FUNCTION_BLOCK Fb_SafetyCheck
VAR_INPUT
END_VAR
VAR_OUTPUT
END_VAR
VAR
	i, j:INT;
	m_checkDelay :ARRAY[1..g_maxNum] OF checkDelay;
	m_checkDelayTime :checkDelayTime;
	m_checkPermit:ARRAY[1..g_maxNum] OF  checkPermit;
	
	m_jntErrFlag:ARRAY[1..g_maxNum,0..g_maxArmJoint,1..3] OF BOOL;
	m_armErrFlag:ARRAY [1..g_maxNum,1..3] OF BOOL;
	m_errCode:UDINT;
	
	
	m_errNumType: ARRAY [1..3] OF INT;
	m_ArrayErrCodeType:ARRAY [1..3] OF ARRAY [0..100] OF UDINT;
	
	//The fault is sent to the UI at the frequency of 0.1S
	m_errCodeUpdateFlag: ARRAY [1..3] OF BOOL;
	m_errCodeUpdateTon: ARRAY [1..3] OF TON;
	
	m_curJntTorqueIOlast :ARRAY [1..g_maxArmNum] OF vec7di;  
	m_cmdJntPosLast : ARRAY [1..g_maxArmNum] OF vec7d;  
	m_cartCurJntTorqueIOlast :ARRAY [1..4] OF LREAL;  
	m_cartCmdJntPosLast : ARRAY [1..4] OF LREAL; 
	o_ErrCode:ARRAY [1..3] OF UDINT;
		
	m_PromptMassBusy:BOOL;
	m_PromptFlag:ARRAY[1..g_maxNum,1..20] OF UINT;
	m_deleteCode:UDINT;
	
END_VAR


VAR CONSTANT
	m_codeUpdateDelay:TIME:=T#0.1S;
	
	//Fault level: 1 indicates  prompt message, 2 indicates a recoverable fault and 3 indicates an unrecoverable fault
	m_promptMessageLevel : UINT :=1;
	m_rcvLevel : UINT :=2;
	m_unrcvLevel : UINT :=3;
END_VAR

METHOD armSafetyCheck : BOOL
VAR_INPUT
	i_armId:UDINT;
	i_safetyCheckVar :ARRAY[1..g_maxNum] OF checkInputVariable;
	i_masterJointData : ST_MasterJointData;
END_VAR

VAR
	k:INT;
END_VAR

//驱动器状态监测、驱动器未连接
FOR i:=1 TO g_mJntNum BY 1 DO
	m_checkDelay[i_ArmId].T_jntStatusErr[i](IN:= (i_safetyCheckVar[i_ArmId].m_masterDriverInput[i].m_statusWord=0 AND m_checkPermit[i_ArmId].m_jntStatusErr[i]), PT:=m_checkDelayTime.Ti_jntStatusErr , Q=> , ET=> );
	IF m_checkDelay[i_ArmId].T_jntStatusErr[i].Q  THEN
		errCodeAssign(i_ArmId, i_ArmId,  0, i, 16#3002 ,m_unrcvLevel );
	END_IF
END_FOR



//关节编码器监测
FOR i:=1 TO g_mJntNum BY 1 DO
	m_checkDelay[i_ArmId].T_linkEncErr[i](IN:= (i_safetyCheckVar[i_ArmId].m_masterDriverInput[i].m_linkEncoder=g_maxLinkEnc OR i_safetyCheckVar[i_ArmId].m_masterDriverInput[i].m_linkEncoder=g_minLinkEnc) AND m_checkPermit[i_ArmId].m_linkEncErr[i], PT:=m_checkDelayTime.Ti_linkEncErr , Q=> , ET=> );
	IF m_checkDelay[i_ArmId].T_linkEncErr[i].Q THEN
		errCodeAssign(i_ArmId, i_ArmId,  0, i,  16#3003 ,m_unrcvLevel );
	END_IF
END_FOR


//驱动器错误检测
FOR i:=1 TO g_mJntNum BY 1 DO
	m_checkDelay[i_ArmId].T_DriveErr[i](IN:= (i_safetyCheckVar[i_ArmId].m_masterDriverInput[i].m_driverError AND 16#20)=g_driveErrWord AND m_checkPermit[i_ArmId].m_driveErr[i] , PT:=m_checkDelayTime.Ti_driveErr , Q=> , ET=> );
	IF m_checkDelay[i_ArmId].T_DriveErr[i].Q THEN
		errCodeAssign(i_ArmId, i_ArmId,  0, i, 16#3004 ,m_unrcvLevel );
	END_IF
END_FOR


//双编码器偏差过大检测
FOR i:=1 TO g_mJntNum BY 1 DO
	m_checkDelay[i_ArmId].T_armJntEncErr[i](IN:= ABS(i_masterJointData.m_curLinkPos[i_armId][i]-i_masterJointData.m_curJntPos[i_armId][i])>=g_armMaxJntEncErr[i] AND m_checkPermit[i_ArmId].m_armJntEncErr[i], PT:=m_checkDelayTime.Ti_armJntEncErr , Q=> , ET=> );
	IF m_checkDelay[i_ArmId].T_armJntEncErr[i].Q THEN
		errCodeAssign( i_ArmId, i_ArmId,  0, i, 16#3005, m_unrcvLevel );
	END_IF
END_FOR


//关节运动超限位
FOR i:=1 TO g_mJntNum BY 1 DO
	m_checkDelay[i_armId].T_outOfLimit[i](IN:= i_masterJointData.m_curJntPos[i_armId][i]>= (GVL_ArmJointParameters.g_maxJntPos[i_armId,i] + g_armJntPosLimitBuffer[i]) OR i_masterJointData.m_curJntPos[i_armId][i]<=(GVL_ArmJointParameters.g_minJntPos[i_armId,i] - g_armJntPosLimitBuffer[i]) AND m_checkPermit[i_ArmId].m_outOfLimit[i], PT:=m_checkDelayTime.Ti_outofLimit , Q=> , ET=> );
	IF m_checkDelay[i_armId].T_outOfLimit[i].Q THEN
		errCodeAssign(i_armId, i_ArmId+3,  0, i, 16#3006, m_unrcvLevel );
	END_IF
END_FOR


//驱动器内部通讯错误
FOR i:=1 TO g_mJntNum BY 1 DO
	m_checkDelay[i_armId].T_currentIsNotUpdate[i](IN:= (i_safetyCheckVar[i_ArmId].m_masterDriverInput[i].m_current=m_curJntTorqueIOlast[i_ArmId][i] AND m_checkPermit[i_ArmId].m_currentIsNotUpdate[i]), PT:=m_checkDelayTime.Ti_currentIsNotUpdate , Q=> , ET=> );
	IF  m_checkDelay[i_armId].T_currentIsNotUpdate[i].Q THEN
		errCodeAssign(i_armId, i_ArmId+3,  0, i, 16#3009 ,m_unrcvLevel );
	END_IF
	m_curJntTorqueIOlast[i_armId][i]:=i_safetyCheckVar[i_armId].m_masterDriverInput[i].m_current;
END_FOR


//关节跟随误差过大
FOR i:=1 TO g_mJntNum BY 1 DO
	m_checkDelay[i_ArmId].T_armJntFollowErr[i](IN:= ABS(i_masterJointData.m_cmdJntPos[i_armId][i]- i_masterJointData.m_curJntPos[i_armId][i])>g_armMaxJntFollowErr[i]  AND m_checkPermit[i_ArmId].m_armJntFollowErr[i], PT:=m_checkDelayTime.Ti_armJntFollowErr , Q=> , ET=> );
	IF m_checkDelay[i_ArmId].T_armJntFollowErr[i].Q THEN
		errCodeAssign(i_ArmId, i_ArmId+3,  0, i, 16#2002, m_rcvLevel );
	END_IF
END_FOR


//关节速度监控
//FOR i:=1 TO g_mJntNum BY 1 DO
//	m_checkDelay[i_ArmId].T_jntVelErr[i](IN:= ABS (i_masterJointData.m_curJntVel[i_armId][i])>g_safetyJntVel[i+g_setupJntNum] AND m_checkPermit[i_ArmId].m_jntVelErr[i], PT:=m_checkDelayTime.Ti_jntVelErr , Q=> , ET=> );
//	IF m_checkDelay[i_ArmId].T_jntVelErr[i].Q THEN
//		errCodeAssign(i_ArmId, i_ArmId+3,  0, i, 16#2003, m_rcvLevel );
//	END_IF
//END_FOR


//笛卡尔空间指令与位置偏差检测
//FOR i:=1 TO 6 BY 1 DO
//	m_checkDelay[i_ArmId].T_spacePoseErr[i](IN:= i_safetyCheckVar[i_ArmId].m_spacePoseErr[i]> g_maxCartPoseErr[i] AND m_checkPermit[i_ArmId].m_spacePoseErr[i], PT:=m_checkDelayTime.Ti_spacePoseErr , Q=> , ET=> );
//	IF m_checkDelay[i_ArmId].T_spacePoseErr[i].Q THEN
//		errCodeAssign(i_ArmId, i_ArmId+3, 1, i, 16#2004, m_rcvLevel );
//	END_IF
//END_FOR


//电流超限监测
FOR i:=1 TO g_mJntNum BY 1 DO
	m_checkDelay[i_armId].T_jntCurrentErr[i](IN:= ABS(i_safetyCheckVar[i_armId].m_motorCurrentIntegral[i])>g_motorCurrentLimit[i] AND m_checkPermit[i_ArmId].m_jntCurrentErr[i], PT:=m_checkDelayTime.Ti_jntCurrentErr , Q=> , ET=> );
	IF m_checkDelay[i_armId].T_jntCurrentErr[i].Q THEN
		errCodeAssign(i_armId, i_ArmId+3,  0, i, 16#2005, m_rcvLevel );
	END_IF
END_FOR


//Ethercat通讯检测
FOR i:=1 TO g_mJntNum BY 1 DO
	IF NOT i_safetyCheckVar[i_ArmId].m_EtherCATState[i].EtherCATState THEN
		errCodeAssign(i_ArmId, i_ArmId+3, 0, i, 16#2006, m_rcvLevel );
	END_IF
END_FOR


//自检未完成
IF i_safetyCheckVar[i_armId].m_selfCheckFail[i] THEN
	errCodeAssign(i_armId, i_ArmId+3,  0, i, 16#2008, m_rcvLevel );
END_IF
END_METHOD

METHOD arrayDeleteFrist : ARRAY [0..100] OF UDINT;
VAR_INPUT
	i_array:ARRAY [0..100] OF UDINT;
END_VAR

VAR
	k:INT;
END_VAR

arrayDeleteFrist[100]:=0;

FOR k:=0 TO 99 BY 1 DO
	arrayDeleteFrist[k]:=i_array[k+1];
END_FOR
END_METHOD

METHOD arrayDeleteInput : BOOL
VAR_INPUT
	i_Array:ARRAY[0..100] OF UDINT;
	i_DeleteCode:UDINT;
END_VAR

VAR_OUTPUT
	o_Array:ARRAY[0..100] OF UDINT;
	
END_VAR

VAR
	i:INT;
	Falg:BOOL;
END_VAR

FOR i:=0 TO 20 BY 1 DO 
	IF i_Array[i]=i_DeleteCode THEN
		Falg:=TRUE;
	END_IF
	
	IF Falg=TRUE THEN
		o_Array[i]:=i_Array[i+1];
	ELSE
		o_Array[i]:=i_Array[i];
	END_IF
END_FOR
o_Array[20]:=0;
END_METHOD

METHOD arrayFIFO : ARRAY [0..100] OF  UDINT
VAR_INPUT
	i_array:ARRAY[0..100] OF UDINT;
	i_newData:UDINT;
END_VAR

VAR
	i:INT;
END_VAR

FOR i:=0 TO 20 BY 1 DO
	arrayFIFO[i+1]:=i_array[i];
END_FOR

arrayFIFO[0]:=i_newData;
END_METHOD

METHOD arrayFILO : ARRAY [0..100] OF  UDINT
VAR_INPUT
	i_array:ARRAY[0..100] OF UDINT;
	i_newData:UDINT;
END_VAR

VAR
	i:INT;
END_VAR

FOR i:=0 TO 20 BY 1 DO
	arrayFILO[i]:=i_array[i];
	IF i_array[i]=0 THEN
		arrayFILO[i]:=i_newData;
		EXIT;
	END_IF
END_FOR
END_METHOD

METHOD cartSafetyCheck : BOOL
VAR_INPUT
	i_armId:UDINT;
	i_safetyCheckVar : checkInputVariable;
	i_cartJointData : ST_CartJointData;
END_VAR


VAR
	k:INT;
END_VAR


//驱动器状态监测、驱动器未连接
FOR i:=1 TO g_maxCartJoint BY 1 DO
	m_checkDelay[i_armId].T_cartJntStatusErr[i](IN:= (i_safetyCheckVar.m_cartDriverInput[i].m_statusWord=0 AND m_checkPermit[i_ArmId].m_cartJntStatus[i]), PT:=m_checkDelayTime.Ti_CarJntStatus , Q=> , ET=> );
	IF m_checkDelay[i_armId].T_cartJntStatusErr[i].Q THEN
		errCodeAssign(i_armId, i_ArmId+3,  0, i, 16#3002 ,m_unrcvLevel );
	END_IF
END_FOR



//关节编码器监测
FOR i:=1 TO g_maxCartJoint BY 1 DO
	m_checkDelay[i_armId].T_cartLinkEncErr[i](IN:= (i_safetyCheckVar.m_cartDriverInput[i].m_linkEncoder=g_cartMaxLinkEnc[i] OR i_safetyCheckVar.m_cartDriverInput[i].m_linkEncoder=g_cartMinLinkEnc[i]) AND m_checkPermit[i_ArmId].m_cartJntEncErr[i], PT:=m_checkDelayTime.Ti_CarActSec , Q=> , ET=> );
	IF m_checkDelay[i_armId].T_cartLinkEncErr[i].Q THEN
		errCodeAssign(i_armId, i_ArmId+3,  0, i, 16#3003 ,m_unrcvLevel );
	END_IF
END_FOR


//驱动器错误检测
FOR i:=1 TO g_maxCartJoint BY 1 DO
	m_checkDelay[i_armId].T_cartDriveErr[i](IN:= (i_safetyCheckVar.m_cartDriverInput[i].m_driverError AND 16#20)=32 AND m_checkPermit[i_ArmId].m_cartDriveErr[i] , PT:=m_checkDelayTime.Ti_CarDriveErr , Q=> , ET=> );
	IF m_checkDelay[i_armId].T_cartDriveErr[i].Q THEN
		errCodeAssign(i_armId, i_ArmId+3,  0, i, 16#3004 ,m_unrcvLevel );
	END_IF
END_FOR



//台车双编码器偏差过大
FOR i:=1 TO g_maxCartJoint BY 1 DO
	m_checkDelay[i_armId].T_cartJntEncErr[i](IN:= ABS (i_cartJointData.m_curLinkPos[i]-i_cartJointData.m_curJntPos[i])>g_cartMaxJntEncErr[i] AND m_checkPermit[i_ArmId].m_cartJntEncErr[i], PT:=m_checkDelayTime.Ti_CarDualEncDev , Q=> , ET=> );
	IF m_checkDelay[i_armId].T_cartJntEncErr[i].Q THEN
		errCodeAssign(i_armId, i_ArmId+3,  0, i, 16#3005 ,m_unrcvLevel );
	END_IF
END_FOR


//关节运动超限位
FOR i:=1 TO g_maxCartJoint BY 1 DO
	m_checkDelay[i_armId].T_cartOutOfLimit[i](IN:= (i_cartJointData.m_curJntPos[i]>=g_cartMaxJntLimit[i] OR i_cartJointData.m_curJntPos[i]<=g_cartMinJntLimit[i]) AND m_checkPermit[i_ArmId].m_cartOutOfLimit[i] , PT:=m_checkDelayTime.Ti_CaroutofLimit , Q=> , ET=> );
	IF m_checkDelay[i_armId].T_cartOutOfLimit[i].Q THEN
		errCodeAssign(i_armId, i_ArmId+3,  0, i, 16#3006 ,m_unrcvLevel );
	END_IF
END_FOR


//驱动器内部通讯错误
FOR i:=1 TO g_maxCartJoint BY 1 DO
	m_checkDelay[i_armId].T_cartCurrentIsNotUpdate[i](IN:= (i_safetyCheckVar.m_cartDriverInput[i].m_current=m_cartCurJntTorqueIOlast[i] AND m_checkPermit[i_ArmId].m_cartCurrentIsNotUpdate[i]), PT:=m_checkDelayTime.Ti_CarTorMotor , Q=> , ET=> );
	IF m_checkDelay[i_armId].T_cartCurrentIsNotUpdate[i].Q THEN
		errCodeAssign(i_armId, i_ArmId+3,  0, i, 16#3009 ,m_unrcvLevel );
	END_IF
	m_cartCurJntTorqueIOlast[i]:=i_safetyCheckVar.m_cartDriverInput[i].m_current;
END_FOR


//StopButton
IF NOT i_safetyCheckVar.SlaveStopButton OR i_safetyCheckVar.PCStopButton=0 OR i_safetyCheckVar.MasterStopButton THEN
	errCodeAssign(i_armId, 16#FF, 0, 0, 16#2001, m_rcvLevel );
END_IF


//关节跟随误差过大
FOR i:=1 TO g_maxCartJoint BY 1 DO
	m_checkDelay[i_armId].T_cartJntFollowErr[i](IN:= ABS(i_cartJointData.m_cmdJntPos[i]- i_cartJointData.m_curJntPos[i])>g_cartMaxJntFollowErr[i]  AND m_checkPermit[i_ArmId].m_cartFollowErr[i], PT:=m_checkDelayTime.Ti_CarFollowDev , Q=> , ET=> );
	IF m_checkDelay[i_armId].T_cartJntFollowErr[i].Q THEN
		errCodeAssign(i_armId, i_ArmId+3,  0, i, 16#2002 ,m_rcvLevel );
	END_IF
END_FOR


//关节速度监控
FOR i:=1 TO g_maxCartJoint BY 1 DO
	m_checkDelay[i_armId].T_cartJntVelErr[i](IN:= ABS(i_cartJointData.m_curJntVel[i])>g_cartMaxJntVel[i] AND m_checkPermit[i_ArmId].m_cartJntVelErr[i], PT:=m_checkDelayTime.Ti_CarJntVel , Q=> , ET=> );
	IF m_checkDelay[i_armId].T_cartJntVelErr[i].Q THEN
		errCodeAssign(i_armId, i_ArmId+3,  0, i, 16#2003 ,m_rcvLevel );
	END_IF
END_FOR


//电流超限监测
FOR i:=1 TO g_maxCartJoint BY 1 DO
	m_checkDelay[i_armId].T_cartJntCurrentErr[i](IN:= ABS(i_cartJointData.m_curJntTrq[i])>g_cartMaxJntCurrent[i] AND m_checkPermit[i_ArmId].m_cartJntCurrentErr[i], PT:=m_checkDelayTime.Ti_CarJntCurrent , Q=> , ET=> );
	IF m_checkDelay[i_armId].T_cartJntCurrentErr[i].Q THEN
		errCodeAssign(i_armId, i_ArmId+3,  0, i, 16#2005 ,m_rcvLevel );
	END_IF
END_FOR


//Ethercat通讯检测
FOR i:=1 TO g_maxCartJoint BY 1 DO
	IF NOT i_safetyCheckVar.m_cartEtherCATState[i].EtherCATState THEN
		errCodeAssign(i_armId, i_ArmId+3,  0, i, 16#2006 ,m_rcvLevel );
	END_IF
END_FOR
END_METHOD

PROPERTY checkPermit : REFERENCE TO ARRAY[1..g_maxNum] OF  checkPermit
GET
checkPermit ref= m_checkPermit;
END_GET
SET
END_SET
END_PROPERTY

METHOD electriAngleDev : DINT
VAR_INPUT
	i_motorElectriAngleDev : DINT;
END_VAR

IF i_motorElectriAngleDev > 50000 THEN
	electriAngleDev := i_motorElectriAngleDev - 65535;
ELSIF i_motorElectriAngleDev < -50000 THEN
	electriAngleDev := i_motorElectriAngleDev + 65535;
ELSE
	electriAngleDev := i_motorElectriAngleDev;
END_IF
END_METHOD

METHOD errCodeAssign : BOOL
VAR_INPUT
	i_armId:UDINT;
	i_errLocation:UDINT;
	i_errCodeMode:UDINT;
	i_errJoint:UDINT;
	i_errID:UDINT;
	i_errFlagID :UINT;
END_VAR
IF m_jntErrFlag[i_armId,i_errJoint,i_errFlagID]=FALSE THEN
	m_jntErrFlag[i_armId,i_errJoint,i_errFlagID]:=TRUE;
	m_errCode:=SHL(i_errLocation,24)+SHL(i_errCodeMode,20)+SHL(i_errJoint,16)+i_errID;
	
	
	IF i_errID>=16#3000 THEN
		m_errNumType[m_unrcvLevel]:=LIMIT(0,m_errNumType[m_unrcvLevel]+1,100);
		m_arrayErrCodeType[m_unrcvLevel][m_errNumType[m_unrcvLevel]]:=m_errCode;
		g_arrayErrCodeArm[i_armId]:=arrayFILO(i_Array:= g_arrayErrCodeArm[i_ArmId], i_NewData:=m_errCode );
		m_armErrFlag[i_armId,m_unrcvLevel]:=TRUE;
		
	ELSIF i_errID>=16#2000 THEN
		m_errNumType[m_rcvLevel]:=LIMIT(0,m_errNumType[m_rcvLevel]+1,100);
		m_arrayErrCodeType[m_rcvLevel][m_errNumType[m_rcvLevel]]:=m_errCode;
		g_arrayErrCodeArm[i_armId]:=arrayFILO(i_Array:= g_arrayErrCodeArm[i_ArmId], i_NewData:=m_errCode );
		m_armErrFlag[i_armId,m_rcvLevel]:=TRUE;
		
	END_IF
END_IF
END_METHOD

METHOD errCodeUpdating :ARRAY [1..3] OF UDINT;
VAR_INPUT
END_VAR

m_errCodeUpdateTon[m_unrcvLevel](IN:= NOT m_errCodeUpdateFlag[3], PT:=m_codeUpdateDelay , Q=> m_errCodeUpdateFlag[3], ET=> );
IF m_errCodeUpdateFlag[m_unrcvLevel] THEN
	IF m_errNumType[m_unrcvLevel]>=1 THEN
		m_ArrayErrCodeType[m_unrcvLevel]:=ArrayDeleteFrist(i_Array:=m_ArrayErrCodeType[3]) ;
		o_ErrCode[m_unrcvLevel]:=m_ArrayErrCodeType[m_unrcvLevel][0] ;
		m_errNumType[m_unrcvLevel]:=m_errNumType[m_unrcvLevel]-1;
	END_IF
END_IF


m_errCodeUpdateTon[m_rcvLevel](IN:= NOT m_errCodeUpdateFlag[2], PT:=m_codeUpdateDelay , Q=> m_errCodeUpdateFlag[2], ET=> );
IF m_errCodeUpdateFlag[m_rcvLevel] THEN
	IF m_errNumType[m_rcvLevel]>=1 THEN
		m_ArrayErrCodeType[m_rcvLevel]:=ArrayDeleteFrist(i_Array:=m_ArrayErrCodeType[m_rcvLevel]) ;
		o_ErrCode[m_rcvLevel]:=m_ArrayErrCodeType[m_rcvLevel][0] ;
		m_errNumType[m_rcvLevel]:=m_errNumType[m_rcvLevel]-1;
	END_IF
END_IF
END_METHOD

METHOD errFlagReset : BOOL
VAR_INPUT
END_VAR

FOR i := 1 TO g_maxArmNum DO
	FOR j :=0 TO g_maxArmJoint DO
		m_jntErrFlag[i, j, 2]:=FALSE;
	END_FOR
	m_armErrFlag[i, 2]:=FALSE;
END_FOR

o_ErrCode[2]:=0;
END_METHOD

METHOD poseErrCheck : vec6d
VAR_INPUT
	i_cmdPose : ST_Frame;
	i_curPose :ST_Frame;
END_VAR

VAR
	posErr,oriErr:Vec3d;
	matT,rotErr:Mat3d;
	errAngle :LREAL;
	errAxis :Vec3d;
	i : INT;
END_VAR
vecSub(i_cmdPose.m_pos, i_curPose.m_pos,posErr);

matTranspose(i_cmdPose.m_rot, matT);
matMultiply(matT,i_curPose.m_rot, rotErr);
rot2AngAxis(rotErr, angle=>errAngle, axis=>errAxis);
vecMultiNum(errAxis, errAngle,oriErr);

FOR i := 1 TO 6 DO
	IF i <= 3 THEN
		poseErrCheck[i] := posErr[i];
	ELSE
		poseErrCheck[i] := oriErr[i];
	END_IF
END_FOR
END_METHOD

METHOD promptMassCode : BOOL
VAR_INPUT
	i_PromptStatus:BOOL;
	i_ArmId:UDINT;
	i_ErrID:UDINT;
	i_ErrLocation:UDINT;
END_VAR

m_PromptMassBusy:=TRUE;

//提示置位
IF i_PromptStatus=TRUE AND m_PromptFlag[i_ArmId,i_ErrID]=0 THEN
	m_PromptFlag[i_ArmId,i_ErrID]:=1;
END_IF

//输出提示故障码
IF m_PromptFlag[i_ArmId,i_ErrID]=1 THEN
	m_ErrCode:=SHL(i_ErrLocation,24)+SHL(0,20)+SHL(0,16)+i_ErrID+16#1010;
	//m_ErrNumType1:=LIMIT(0,m_ErrNumType1+1,100);
	m_ArrayErrCodeType[1]:=ArrayFIFO(i_Array:= m_ArrayErrCodeType[1], i_NewData:=m_ErrCode );//m_ErrCode;
	m_PromptFlag[i_ArmId,i_ErrID]:=2;
END_IF

//清除提示故障码
IF m_PromptFlag[i_ArmId,i_ErrID]=2 AND i_PromptStatus=FALSE THEN
	m_deleteCode:=SHL(i_ErrLocation,24)+SHL(0,20)+SHL(0,16)+i_ErrID+16#1020;
	ArrayDeleteInput(i_Array:= m_ArrayErrCodeType[1], i_DeleteCode:=m_deleteCode , o_Array=> m_ArrayErrCodeType[1]);
	//m_ErrNumType1:=m_ErrNumType1-1;
	m_PromptFlag[i_ArmId,i_ErrID]:=0;
END_IF
o_ErrCode[1]:=m_ArrayErrCodeType[1][0];
m_PromptMassBusy:=FALSE;
END_METHOD

METHOD systemSafetyCheck : BOOL
VAR_INPUT
	i_armId:UDINT;
	i_safetyCheckVar :ARRAY[1..g_maxNum] OF checkInputVariable;
	i_cartJointData : ST_CartJointData;
	i_masterJointData : ST_MasterJointData;
END_VAR

VAR
	k:INT;
END_VAR

IF i_armId =g_cartNum THEN 
	//cart safrty check
	cartSafetyCheck(i_armId,i_safetyCheckVar[i_armId],i_cartJointData);
ELSE
	//master arms safety check
	armSafetyCheck(i_armId,i_safetyCheckVar,i_masterJointData);
	
	//StopButton
	IF NOT i_safetyCheckVar[i_ArmId].SlaveStopButton OR i_safetyCheckVar[i_ArmId].PCStopButton=0 OR i_safetyCheckVar[i_ArmId].MasterStopButton THEN
		errCodeAssign(i_ArmId, 16#0C, 0, 0, 16#2001, m_rcvLevel );
	END_IF
END_IF


//prompt message
FOR i:=1 TO 20 BY 1 DO
	PromptMassCode( i_safetyCheckVar[i_ArmId].m_promptStatus[i], i_ArmId,  i,  i_safetyCheckVar[i_ArmId].m_promptLocation[i]);
END_FOR
END_METHOD

END_FUNCTION_BLOCK

(* stored: Version 1.1.0.1, ProductVersion 3.1.4024.11
   POU Fb_SafetyCheck: Id {d7e5b419-2971-4dae-96a7-39fe3a1a6245}, SpecialFunc None
   Folder interface: Id {17cc820b-439e-4bcd-b035-470b65e01b6b}
   Method armSafetyCheck: Id {1102e175-6107-4706-a6ad-ea5e8fc76a1b}
   Method arrayDeleteFrist: Id {00e49c9f-cbe8-4b26-b05a-c4b6acb31969}
   Method arrayDeleteInput: Id {980f1673-9d6d-4af2-a068-78f386b10642}
   Method arrayFIFO: Id {655e2224-db9d-4b4a-8461-cda6c8a0a0dc}
   Method arrayFILO: Id {26262d95-ef1c-497d-b548-c28fcd1771c9}
   Method cartSafetyCheck: Id {64489d60-54d3-406d-a82e-df5d6a98f0f1}
   Property checkPermit: Id {4ac5d9ef-e4e1-4258-a3b3-a263171adb15}
   Get Get: Id {5a600670-0a2f-4560-9a82-9a30fff97e6d}
   Set Set: Id {06536298-2ca0-4bed-b4ee-b29089d28252}
   Method electriAngleDev: Id {8c2ea40a-ba18-4d9e-8d1f-4ea5c9f320b3}
   Method errCodeAssign: Id {c6bfedc5-fddc-4db6-ba7d-64971d20a433}
   Method errCodeUpdating: Id {0b3c9bb2-9217-4fc9-b998-e4a685172889}
   Method errFlagReset: Id {2f8c115b-de2b-4c35-92d2-fdbed32dcf1f}
   Method poseErrCheck: Id {634b1f68-028c-4865-89df-6d37274cf53c}
   Method promptMassCode: Id {97898266-aa01-4d86-bccd-f23152d91670}
   Method systemSafetyCheck: Id {7874ef26-88d5-4eb7-8db9-4fa17a2dd1f0} *)
